(* IEC 61131-3 sources: volt/packages/volt-lsp-iec/test-corpus/lenze-mid/Device/Plc Logic/Application/Library Manager/CAA CANopen Manager, 14 files *)

(* ---- ERROR.dut ---- *)
TYPE ERROR :
(
	NO_ERROR := 0,
	FIRST_ERROR := 10300,
	TIME_OUT := 10301,
	NO_MORE_MEMORY := 10302,
	INVALID_HANDLE := 10303,
	WRONG_PARAMETER := 10304,
	NODEID_UNKNOWN := 10305,
	NETID_UNKNOWN := 10306,
	NETID_OCCUPIED := 10307,
	FIRST_MF := 10349,
	LAST_ERROR := 10399
);
END_TYPE

(* ---- CANOPENMANAGERVARIABLES.gvl ---- *)
VAR_GLOBAL
	GC_USIMAXNETID : USINT := 9;
	M_ISTACK : ARRAY [0..gc_usiMaxNetId] OF CS.ICanOpenStack;
END_VAR

(* ---- PROPERTYCONSTANTS.gvl ---- *)
VAR_GLOBAL
	GC_UIMAXNETID : UINT := 1;
END_VAR

(* ---- VERSIONCONSTANTS.gvl ---- *)
VAR_GLOBAL
	GC_BYVERSION : BYTE := 1;
	GC_BYVERSION_1 : BYTE := 0;
END_VAR

(* ---- GETPROPERTY.pou ---- *)
FUNCTION GETPROPERTY : UDINT
VAR_INPUT
	UIPROPERTY : UINT;
END_VAR
END_FUNCTION

(* ---- GETSUPPLIERVERSION.pou ---- *)
FUNCTION GETSUPPLIERVERSION : WORD
VAR_INPUT
	XDUMMY : BOOL;
END_VAR
END_FUNCTION

(* ---- SDOABORT.pou ---- *)
FUNCTION SDOABORT : CS.PROC_STATE
VAR_INPUT
	ECMD : CS.PROC_CMD;
	USINETID : USINT;
	PPARAM : POINTER TO CS.SDO_ABORT;
END_VAR
VAR_OUTPUT
	EERROR : CS.ERROR;
END_VAR
END_FUNCTION

(* ---- SDOREAD.pou ---- *)
FUNCTION SDOREAD : CS.PROC_STATE
VAR_INPUT
	ECMD : CS.PROC_CMD;
	USINETID : USINT;
	PPARAM : POINTER TO CS.SDO_READ;
END_VAR
VAR_OUTPUT
	EERROR : CS.ERROR;
END_VAR
END_FUNCTION

(* ---- SDOWRITE.pou ---- *)
FUNCTION SDOWRITE : CS.PROC_STATE
VAR_INPUT
	ECMD : CS.PROC_CMD;
	USINETID : USINT;
	PPARAM : POINTER TO CS.SDO_WRITE;
END_VAR
VAR_OUTPUT
	EERROR : CS.ERROR;
END_VAR
END_FUNCTION

(* ---- STKCLOSE.pou ---- *)
FUNCTION STKCLOSE : CS.PROC_STATE
VAR_INPUT
	ECMD : CS.PROC_CMD;
	USINETID : USINT;
END_VAR
VAR_OUTPUT
	EERROR : CS.ERROR;
END_VAR
END_FUNCTION

(* ---- STKGETINFO.pou ---- *)
FUNCTION STKGETINFO : CS.PROC_STATE
VAR_INPUT
	ECMD : CS.PROC_CMD;
	USINETID : USINT;
	PSTKINFO : POINTER TO CS.STK_INFO;
	PNETINFO : POINTER TO CS.NET_INFO;
END_VAR
VAR_OUTPUT
	EERROR : CS.ERROR;
END_VAR
END_FUNCTION

(* ---- STKOPEN.pou ---- *)
FUNCTION STKOPEN : CS.PROC_STATE
VAR_INPUT
	ECMD : CS.PROC_CMD;
	USINETID : USINT;
	USINODEID : USINT;
	UIBAUDRATE : UINT;
	ESPEC : CS.STK_SPEC;
END_VAR
VAR_OUTPUT
	EERROR : CS.ERROR;
END_VAR
END_FUNCTION

(* ---- STKREGISTER.pou ---- *)
FUNCTION STKREGISTER : CAA.HANDLE
VAR_INPUT
	USINETID : USINT;
	ISTACK : CS.ICanOpenStack;
END_VAR
VAR_OUTPUT
	EERROR : ERROR;
END_VAR
END_FUNCTION

(* ---- STKUNREGISTER.pou ---- *)
FUNCTION STKUNREGISTER : ERROR
VAR_INPUT
	HSTACK : CAA.HANDLE;
END_VAR
END_FUNCTION
